Fanuc KAREL source: kt00302.KL

-- PROVISIONAL review KL for V770-1; original PC SHA256 21408ec40cebc0749cf490e46fdce0527d3827d8df16ddf28878d122dd87b8d1
-- Incomplete behavior may be omitted. Consult companion uncertainty JSON. Do not deploy.
PROGRAM KT00302
%NOLOCKGROUP
VAR
  S1 : STRING[80]
  S2 : STRING[80]
  OUT : BOOLEAN
BEGIN
  -- UNRESOLVED_PC offsets 5-14; opcodes 3F,75
  -- UNRESOLVED_PC offsets 19-28; opcodes 3F,75
  -- UNRESOLVED_PC offsets 33-42; opcodes 3F,75
  -- UNRESOLVED_PC offsets 47-56; opcodes 3F,75
  -- UNRESOLVED_PC offsets 61-80; opcodes 73,73,84,23
  -- UNRESOLVED_PC offsets 85-89; opcodes 7F
END KT00302
